// SIMATIC S7-200 project (STEP 7-Micro/WIN), CPU 216 REL 01.02

SYMBOL_TABLE SYM1
Always_On        SM0.0    // This bit is always on.
First_Scan_On    SM0.1    // This bit is on for the first scan cycle only.
Pot0_Value       SMB28    // Stores value entered by analog adjustment 0. Updated once per cycle in STOP/RUN
Pot1_Value       SMB29    // Stores value entered by analog adjustment 1. Updated once per cycle in STOP/RUN
Run_Compare      M0.0     // Memory bit must be set to compare the average value to upper and lower limits.
END_SYMBOL_TABLE

ORGANIZATION_BLOCK OB_1:OB1
TITLE=
BEGIN
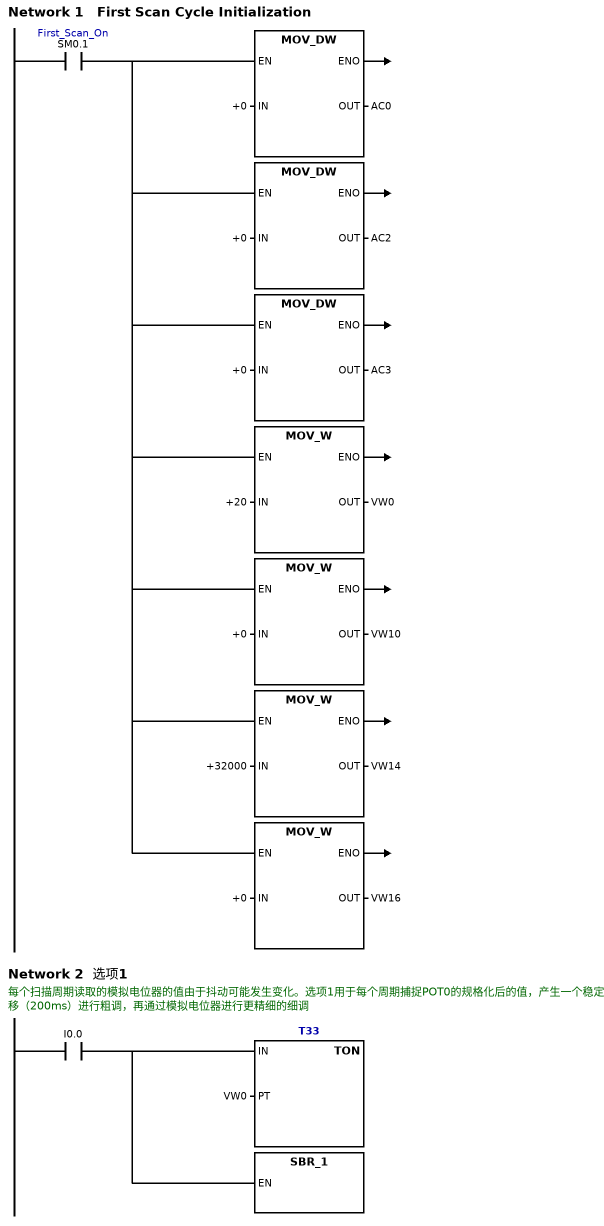
Network 1 //  First Scan Cycle Initialization
// Load S0.1.
// Clear accumulator AC0.
// Clear accumulator AC2.
// Clear accumulator AC3.
// Store value to be used
// with timer T33.
// Set the scan counter to 0.
// Reset lower limit
// workspace.
// Reset upper limit
// workspace.
LD     First_Scan_On:SM0.1
MOVD   +0, AC0
MOVD   +0, AC2
MOVD   +0, AC3
MOVW   +20, VW0
MOVW   +0, VW10
MOVW   +32000, VW14
MOVW   +0, VW16
Network 2 // 选项1
// 每个扫描周期读取的模拟电位器的值由于抖动可能发生变化。选项1用于每个周期捕捉POT0的规格化后的值，产生一个稳定的定时值。选项1展示了一个模拟电位器作为一个定时器的精细调谐器：使用SMB28，通过程序中的偏移（200ms）进行粗调，再通过模拟电位器进行更精细的细调
// Load input I0.0.
// Enable timer T33, with PT
// from VW0.
// Call SBR1.
LD     I0.0
TON    T33, VW0
CALL   SBR_1:SBR1
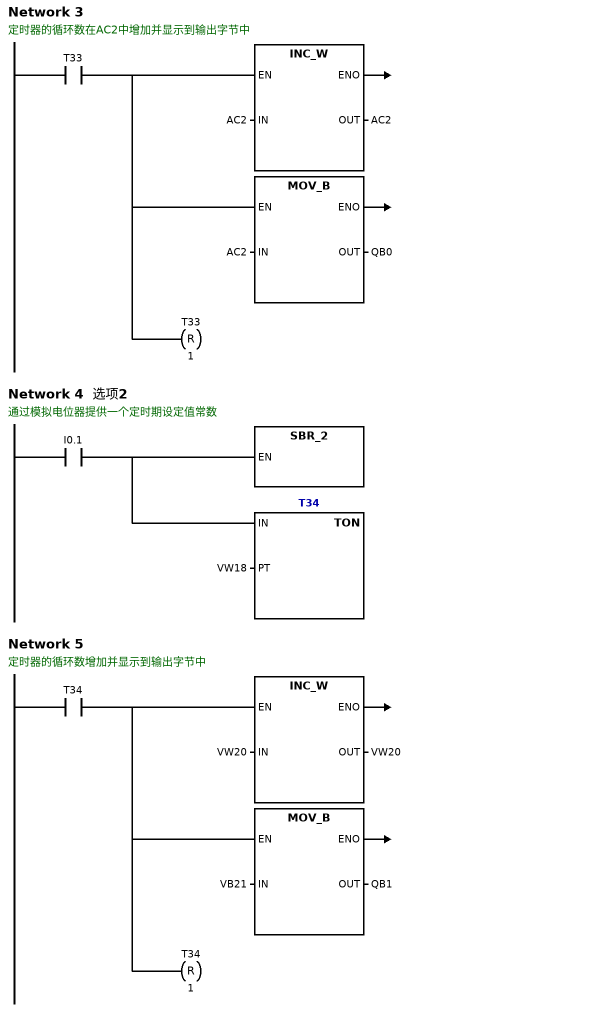
Network 3
// 定时器的循环数在AC2中增加并显示到输出字节中
// Load timer T33.
// Increment the value of
// accumulator AC2 by 1.
// Display the current value
// at the output.
// Reset timer T33.
LD     T33
INCW   AC2
MOVB   AC2, QB0
R      T33, 1
Network 4 // 选项2
// 通过模拟电位器提供一个定时期设定值常数
// Load input I0.1.
// Call SBR2.
// Enable timer T34, with PT
// from VW18.
LD     I0.1
CALL   SBR_2:SBR2
TON    T34, VW18
Network 5
// 定时器的循环数增加并显示到输出字节中
// Load timer T34.
// Increment the value in VW20
// by 1.
// Display the current value of
// VW20 at the output.
// Reset timer T34.
LD     T34
INCW   VW20
MOVB   VB21, QB1
R      T34, 1
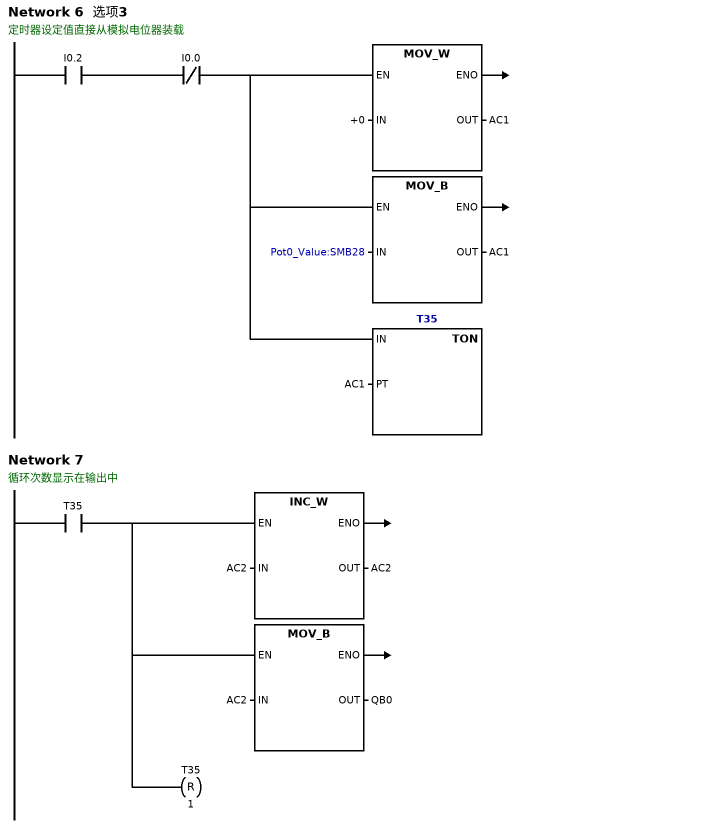
Network 6 // 选项3
// 定时器设定值直接从模拟电位器装载
// Load input I0.2 as a
// Normally Open contact.
// Handle input I0.0 as a
// Normally Closed contact.
// Clear accumulator AC1.
// Load analog adjustment 0
// into accumulator AC1.
// Enable timer T35, with PT
// from AC1.
LD     I0.2
AN     I0.0
MOVW   +0, AC1
MOVB   Pot0_Value:SMB28, AC1
TON    T35, AC1
Network 7
// 循环次数显示在输出中
// Load timer T35.
// Increment the value in AC2
// by 1.
// Display the current value
// of AC2 at the output.
// Reset timer T35.
LD     T35
INCW   AC2
MOVB   AC2, QB0
R      T35, 1
Network 8 //  Main Program End
//  End the main program.
//  MEND					// End the main program.
// 
END_ORGANIZATION_BLOCK

SUBROUTINE_BLOCK SBR_1:SBR1
TITLE=
// ***SUBROUTINES***
// 
// 
BEGIN
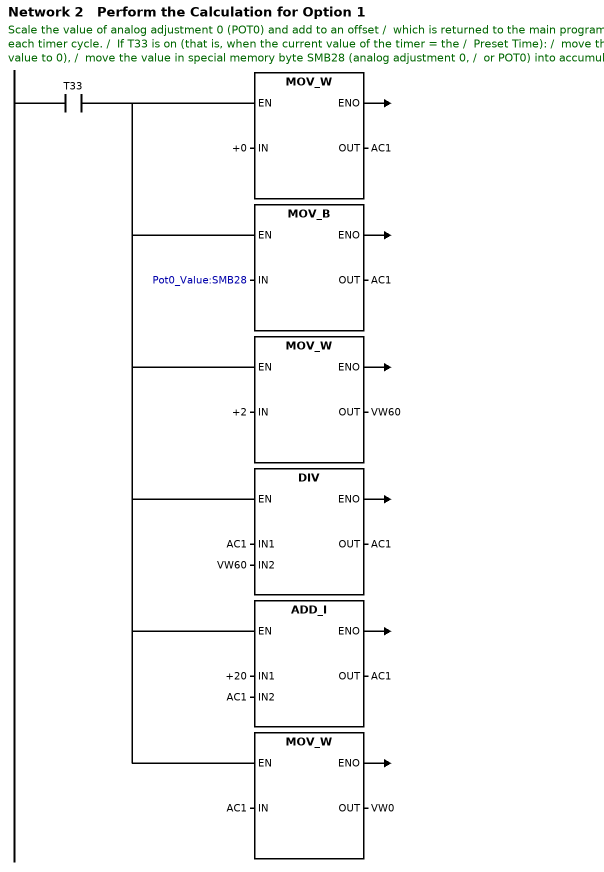
Network 2 //  Perform the Calculation for Option 1
//  Scale the value of analog adjustment 0 (POT0) and add to an offset
//  which is returned to the main program in VW0.
// 
//  Load timer T33 to check for changes to the analog adjustment 0
//  (POT0) each timer cycle.
//  If T33 is on (that is, when the current value of the timer = the
//  Preset Time):
//  move the constant 0 as an input word into accumulator AC1 to
//  clear the accumulator (set its value to 0),
//  move the value in special memory byte SMB28 (analog adjustment 0,
//  or POT0) into accumulator AC1,
//  move the constant 2 as an input word into variable memory word 60
//  (for compatibility with the ladder logic editor),
//  divide the value of analog adjustment 0 by 2 (to scale the
//  potentiometer input range, which is normally from 0 to 255, by
//  one half: that is, to achieve a scaled range of 0 to 127) and put
//  the result in accumulator AC1,
//  add the constant 20 (for the 200-ms offset) to the value in
//  accumulator AC1 and put the result in accumulator AC1 (this will
//  become the new Preset Time for timer T33),
//  and move the value in accumulator AC1 to variable memory word VW0
//  so that the value can be read by means of a programming device.
// 
// Load timer T33.
// Clear accumulator AC1.
// Load analog adjustment 0
// into accumulator AC1.
// Store 2 in VW60.
// Divide the value in AC1 by 2.
// Add an offset of 200 ms.
// Move (copy) the value of
// accumulator AC1 to variable
// memory word VW0.
LD     T33
MOVW   +0, AC1
MOVB   Pot0_Value:SMB28, AC1
MOVW   +2, VW60
DIV    VW60, AC1
+I     +20, AC1
MOVW   AC1, VW0
Network 3 //  End of Subroutine SBR1
//  End SBR1. This instruction returns control to the instruction
//  that follows the CALL instruction for SBR1.
//  RET					// End SBR1.
// 
END_SUBROUTINE_BLOCK

SUBROUTINE_BLOCK SBR_2:SBR2
TITLE=
BEGIN
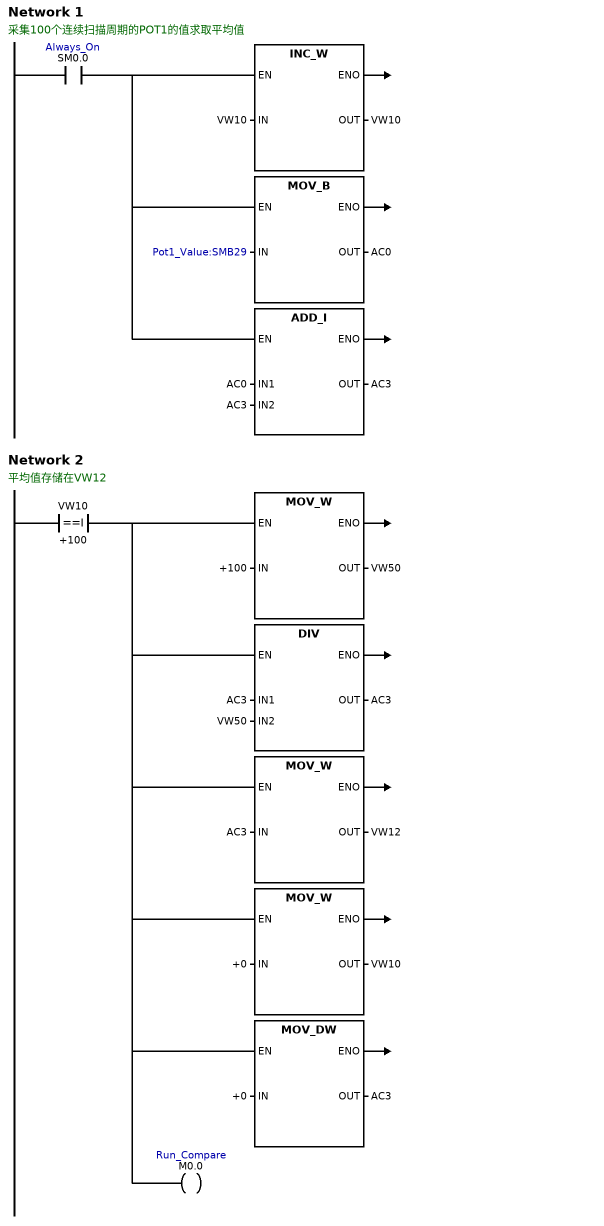
Network 1
// 采集100个连续扫描周期的POT1的值求取平均值
// Load SM0.0.
// Increment the value in VW10
// by 1.
// Load analog adjustment 1 into
// accumulator AC0.
// Add the value in AC0 to the
// value in AC3.
LD     Always_On:SM0.0
INCW   VW10
MOVB   Pot1_Value:SMB29, AC0
+I     AC0, AC3
Network 2
// 平均值存储在VW12
// Compare the value in VW10
// to 100.
// Move 100 into VW50.
// Divide the value in AC3 by 100.
// Store the result in VW12.
// Move 0 into VW10.
// Move 0 as an input double word
// into AC3.
// Turn on M0.0.
LDW=   VW10, +100
MOVW   +100, VW50
DIV    VW50, AC3
MOVW   AC3, VW12
MOVW   +0, VW10
MOVD   +0, AC3
=      Run_Compare:M0.0
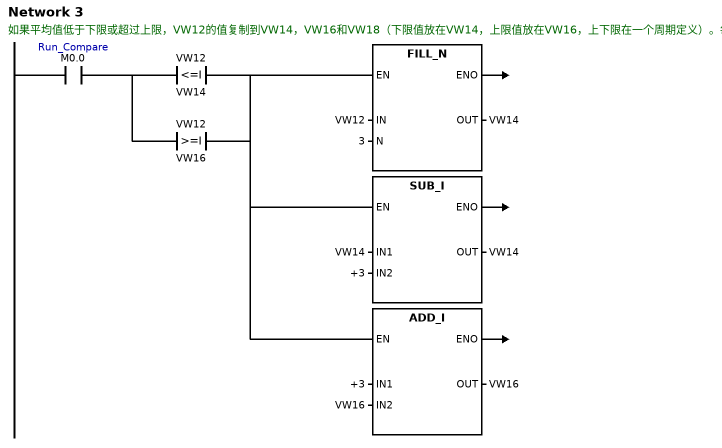
Network 3
// 如果平均值低于下限或超过上限，VW12的值复制到VW14，VW16和VW18（下限值放在VW14，上限值放在VW16，上下限在一个周期定义）。每个限制值与存在VW12的平均值差3ms来确定VW14和VW16的值
// Load M0.0.
// Compare the value in VW12 to
// the value in VW14 for <=.
// Compare the value in VW12 to
// the value in VW16 for >=.
// Combine the values in the
// first and second levels of
// the stack using a logical And
// operation. Load the result to
// the top of the stack.
// Start at VW14 and fill the
// area with the word input
// pattern of VW12 for three
// words.
// Subtract 3 from the value
// in VW14.
// Add 3 to the value in VW16.
LD     Run_Compare:M0.0
LDW<=  VW12, VW14
OW>=   VW12, VW16
ALD
FILL   VW12, VW14, 3
-I     +3, VW14
+I     +3, VW16
Network 4 //  End Subroutine SBR2
//  End SBR2. This instruction returns control to the instruction
//  that follows the CALL instruction for SBR2. This action returns
//  the filtered potentiometer value in variable memory word VW18.
//  RET					// End SBR2.
// 
END_SUBROUTINE_BLOCK
